(* IEC 61131-3 sources: Std_PalletMover/Class/NavigationKinematicPivots, 1 file *)

(* ---- NavigationKinematicPivots.st ---- *)
(*!
<Class
	Name               = "NavigationKinematicPivots"
	Revision           = "0.0"
	RealtimeTask       = "false"
	CyclicTask         = "false"
	BackgroundTask     = "false"
	Sigmatek           = "false"
	OSInterface        = "false"
	HighPriority       = "false"
	Automatic          = "false"
	UpdateMode         = "Prescan"
	SharedCommandTable = "true"
	Objectsize         = "(1140,180)">
	<Channels>
		<Server Name="NumberOfPivotWheels" Visualized="false" Initialize="false" WriteProtected="true" Retentive="false"/>
		<Server Name="ReferenceWheel1" Visualized="false" Initialize="true" WriteProtected="false" Retentive="false"/>
		<Client Name="AGVMode" Required="true" Internal="false"/>
		<Client Name="AgvSettings" Required="true" Internal="false"/>
		<Client Name="ObjKinematicNpivot" Required="true" Internal="true"/>
		<Client Name="objPivotWheel1" Required="false" Internal="false"/>
		<Client Name="objPivotWheel2" Required="false" Internal="false"/>
		<Client Name="objPivotWheel3" Required="false" Internal="false"/>
		<Client Name="objPivotWheel4" Required="false" Internal="false"/>
		<Client Name="objPivotWheel5" Required="false" Internal="false"/>
		<Client Name="objPivotWheel6" Required="false" Internal="false"/>
		<Client Name="objPivotWheel7" Required="false" Internal="false"/>
		<Client Name="objPivotWheel8" Required="false" Internal="false"/>
	</Channels>
	<Network Name="NavigationKinematicPivots">
		<!-- List of Components in this network -->
		<Components>
			<Object
				Name       = "_base"
				Class      = "FunctionBase"
				Position   = "(218,120)"
				Visualized = "false">
				<Channels>
					<Server Name="ObjectStatus"/>
					<Server Name="ToObject"/>
					<Client Name="op_LogData"/>
					<Client Name="p_NextObject"/>
				</Channels>
			</Object>
			<Object
				Name       = "ObjKinematicNpivot"
				Class      = "KinematicNpivot"
				Position   = "(210,360)"
				Visualized = "false">
				<Channels>
					<Server Name="ACTIVATE" Value="1"/>
					<Server Name="ActualTotalDirection"/>
					<Server Name="ActualTotalRadius"/>
					<Server Name="ActualTotalSpeed"/>
					<Server Name="AGVInMotion"/>
					<Server Name="ChaoticManualFrontDirection"/>
					<Server Name="ChaoticManualFrontSpeed"/>
					<Server Name="ChaoticManualRearDirection"/>
					<Server Name="ChaoticManualRearSpeed"/>
					<Server Name="ClassSvr"/>
					<Server Name="Direction"/>
					<Server Name="NumberOfPivotWheels"/>
					<Server Name="Radius"/>
					<Server Name="ReferenceWheel1"/>
					<Server Name="ReferenceWheel2"/>
					<Server Name="Speed"/>
					<Client Name="AGVMode"/>
					<Client Name="chaoticManualModeActive"/>
					<Client Name="objPivotWheel1"/>
					<Client Name="objPivotWheel2"/>
					<Client Name="objPivotWheel3"/>
					<Client Name="objPivotWheel4"/>
					<Client Name="objPivotWheel5"/>
					<Client Name="objPivotWheel6"/>
					<Client Name="objPivotWheel7"/>
					<Client Name="objPivotWheel8"/>
					<Client Name="sigClib"/>
				</Channels>
			</Object>
		</Components>
		<Comments>
		</Comments>
		<!-- List of Connections in this network -->
		<Connections>
			<Connection Source="this.ToObject" Destination="_base.ToObject" Vertices="(1084,210),(804,210),"/>
			<Connection Source="this.ObjectStatus" Destination="_base.ObjectStatus" Vertices="(1084,270),(804,270),"/>
			<Connection Source="this.ObjKinematicNpivot" Destination="ObjKinematicNpivot.ClassSvr"/>
			<Connection Source="_base.p_NextObject" Destination="this.p_NextObject" Vertices="(218,270),(38,270),"/>
			<Connection Source="_base.op_LogData" Destination="this.op_LogData" Vertices="(218,210),(38,210),"/>
			<Connection Source="ObjKinematicNpivot.objPivotWheel1" Destination="this.objPivotWheel1" Vertices="(210,450),(38,390),"/>
			<Connection Source="ObjKinematicNpivot.objPivotWheel2" Destination="this.objPivotWheel2" Vertices="(210,510),(38,450),"/>
			<Connection Source="ObjKinematicNpivot.objPivotWheel3" Destination="this.objPivotWheel3" Vertices="(210,570),(38,510),"/>
			<Connection Source="ObjKinematicNpivot.objPivotWheel4" Destination="this.objPivotWheel4" Vertices="(210,630),(38,570),"/>
			<Connection Source="ObjKinematicNpivot.objPivotWheel5" Destination="this.objPivotWheel5" Vertices="(210,690),(38,630),"/>
			<Connection Source="ObjKinematicNpivot.objPivotWheel6" Destination="this.objPivotWheel6" Vertices="(210,750),(38,690),"/>
			<Connection Source="ObjKinematicNpivot.objPivotWheel7" Destination="this.objPivotWheel7" Vertices="(210,810),(38,750),"/>
			<Connection Source="ObjKinematicNpivot.objPivotWheel8" Destination="this.objPivotWheel8" Vertices="(210,870),(38,810),"/>
			<Connection Source="this.NumberOfPivotWheels" Destination="ObjKinematicNpivot.NumberOfPivotWheels" Vertices="(1084,330),(912,510),"/>
			<Connection Source="this.ReferenceWheel1" Destination="ObjKinematicNpivot.ReferenceWheel1" Vertices="(1084,390),(912,570),"/>
			<Connection Source="ObjKinematicNpivot.AGVMode" Destination="this.AGVMode" Vertices="(210,1050),(38,870),"/>
		</Connections>
		<!-- Headerfiles -->
		<Options>
		</Options>
	</Network>
</Class>
*)
#pragma using FunctionBase

NavigationKinematicPivots : CLASS
: FunctionBase
  //Servers:
	NumberOfPivotWheels 	: SvrCh_DINT;
	ReferenceWheel1 	: SvrCh_DINT;
  //Clients:
	ObjKinematicNpivot 	: CltChCmd_KinematicNpivot;
	AgvSettings 	: CltCh_DINT;
	objPivotWheel1 	: CltChCmd_I_PivotWheel;
	objPivotWheel2 	: CltChCmd_I_PivotWheel;
	objPivotWheel3 	: CltChCmd_I_PivotWheel;
	objPivotWheel4 	: CltChCmd_I_PivotWheel;
	objPivotWheel5 	: CltChCmd_I_PivotWheel;
	objPivotWheel6 	: CltChCmd_I_PivotWheel;
	objPivotWheel7 	: CltChCmd_I_PivotWheel;
	objPivotWheel8 	: CltChCmd_I_PivotWheel;
	AGVMode 	: CltCh_eAGVMode_PTofCls_Standard;
  //Variables:
  //Functions:

	FUNCTION VIRTUAL GLOBAL NumberOfPivotWheels::Read
		VAR_OUTPUT
			output (EAX) 	: DINT;
		END_VAR;

	FUNCTION VIRTUAL GLOBAL ReferenceWheel1::Read
		VAR_OUTPUT
			output (EAX) 	: DINT;
		END_VAR;

	FUNCTION VIRTUAL GLOBAL ReferenceWheel1::Write
		VAR_INPUT
			input (EAX) 	: DINT;
		END_VAR
		VAR_OUTPUT
			result (EAX) 	: DINT;
		END_VAR;
  //Tables:
	FUNCTION @STD
		VAR_OUTPUT
			ret_code	: CONFSTATES;
		END_VAR;
	FUNCTION GLOBAL TAB @CT_;
END_CLASS;

#pragma using KinematicNpivot
#pragma usingLtd I_PivotWheel

FUNCTION VIRTUAL GLOBAL NavigationKinematicPivots::NumberOfPivotWheels::Read
	VAR_OUTPUT
		output (EAX) 	: DINT;
	END_VAR

	NumberOfPivotWheels := ObjKinematicNpivot.NumberOfPivotWheels.Read();
	output := NumberOfPivotWheels;

END_FUNCTION

FUNCTION VIRTUAL GLOBAL NavigationKinematicPivots::ReferenceWheel1::Read
	VAR_OUTPUT
		output (EAX) 	: DINT;
	END_VAR

	ReferenceWheel1 := ObjKinematicNpivot.ReferenceWheel1.Read();
	output := ReferenceWheel1;

END_FUNCTION

FUNCTION VIRTUAL GLOBAL NavigationKinematicPivots::ReferenceWheel1::Write
	VAR_INPUT
		input (EAX) 	: DINT;
	END_VAR
	VAR_OUTPUT
		result (EAX) 	: DINT;
	END_VAR

	ReferenceWheel1 := input;
	result := (ObjKinematicNpivot.ReferenceWheel1.Write(ReferenceWheel1))$DINT;

END_FUNCTION
